TYPE ST_InputsFastDoor :
STRUCT
	HW		: ST_HW_InputsFastDoor; //hardware inputs
END_STRUCT
END_TYPE

(* stored: Version 1.1.0.1, ProductVersion 3.1.4024.9
   DUT ST_InputsFastDoor: Id {c8b80e32-3cbf-4684-968c-2e113a50eb51} *)
